PROGRAM prgLab04_06
VAR
END_VAR

//Primeiro iremos conduzir as comparações básicas

IF GVL.Room1.OccupancySensor THEN
	GVL.Room1.Lighting:=TRUE;
	IF GVL.Room1.Temp > 24 THEN
		GVL.Room1.Heating:=FALSE;
	ELSIF GVL.Room1.Temp <20 THEN
		GVL.Room1.Heating:=TRUE;	
	END_IF
ELSE
	GVL.Room1.Lighting:=GVL.Room1.Heating:=FALSE;	
END_IF
IF GVL.Room1.AirQuality >= GVL.Room1.setpoint THEN
	GVL.Room1.Ventilation:=TRUE;
ELSE
	GVL.Room1.Ventilation:=FALSE;	
END_IF
//Solução lab 06
IF GVL.Room1.Temp< 20 THEN
	GVL.statusRoom1:= E_ROOM_TEMP_STS.baixa;
ELSIF GVL.Room1.Temp >=20 AND GVL.Room1.Temp < 24 THEN
	GVL.statusRoom1:= E_ROOM_TEMP_STS.normal;
ELSIF GVL.Room1.Temp >=24 AND GVL.Room1.Temp < 27 THEN
	GVL.statusRoom1:= E_ROOM_TEMP_STS.moderada;
ELSIF GVL.Room1.Temp >=27 AND GVL.Room1.Temp < 32 THEN
	GVL.statusRoom1:= E_ROOM_TEMP_STS.alta;
ELSIF GVL.Room1.Temp >=32 THEN
	GVL.statusRoom1:= E_ROOM_TEMP_STS.muito_alta;
END_IF

END_PROGRAM

(* stored: Version 1.1.0.1, ProductVersion 3.1.4024.11
   POU prgLab04_06: Id {3badfea7-7024-42bd-8287-83b174bd26b9}, SpecialFunc None *)
